// TIA Portal V20 export
TYPE "F-link_UDT"
// stored: IsFailsafeCompliant true
   STRUCT
      ESTOP_OK : Bool;
      ESTOP_ack_req : Bool;
   END_STRUCT;
END_TYPE
